{attribute 'qualified_only'}
{attribute 'strict'}
{attribute 'to_string'}

TYPE E_EventIDs :
(
	Motor := 0,
	Safety := 1
);
END_TYPE

(* stored: Version 1.1.0.1, ProductVersion 3.1.4024.11
   DUT E_EventIDs: Id {fb131b2a-133e-43df-bcda-6dd200534bb4} *)
